FUNCTION_BLOCK FB_TriggerManagerTestDouble IMPLEMENTS I_TriggerManager
VAR_INPUT
END_VAR
VAR_OUTPUT
END_VAR
VAR
END_VAR

{warning 'Add method implementation '}
METHOD GetAndResetTrigger
VAR_OUTPUT
    bLatchDetected	: BOOL;
    (* [ns]*)
    nLatchTime_ns	: ULINT;
END_VAR
END_METHOD

END_FUNCTION_BLOCK

(* stored: Version 1.1.0.1
   POU FB_TriggerManagerTestDouble: Id {83d68cdb-b331-4489-93e7-4f577042af13}, SpecialFunc None
   Method GetAndResetTrigger: Id {1a41ea64-f5bb-4476-a132-a58d8941b58e} *)
